// SIMATIC S7-200 SMART project (STEP 7-Micro/WIN SMART), CPU SR20

SYMBOL_TABLE 表格 1
搅拌1T定时器          C0
循环定时器            C1
任务阶段             VW10     // 当前任务阶段
提示注肥量            VW12
搅拌时长1T           VW14
目标液位1T           VW16     // 1T注水液位
当前液位1T           VW18
目标液位3T           VW20
当前液位3T           VW22
循环时长             VW24
运输完成标志1T到3T      VW26     // 启动运输前需要上位机置0
循环完成标志           VW28     // 循环前需要上位机清零
排污完成标志           VW30     // 排污前需要上位机清零
排污时长             VW32
水表               VW34
END_SYMBOL_TABLE

SYMBOL_TABLE 系统符号
Always_On        SM0.0    // 始终接通
First_Scan_On    SM0.1    // 仅在第一个扫描周期时接通
Clock_60s        SM0.4    // 针对 1 分钟的周期时间，时钟脉冲接通 30 s，断开 30 s.
END_SYMBOL_TABLE

ORGANIZATION_BLOCK MAIN:OB1
TITLE=注肥功能
BEGIN
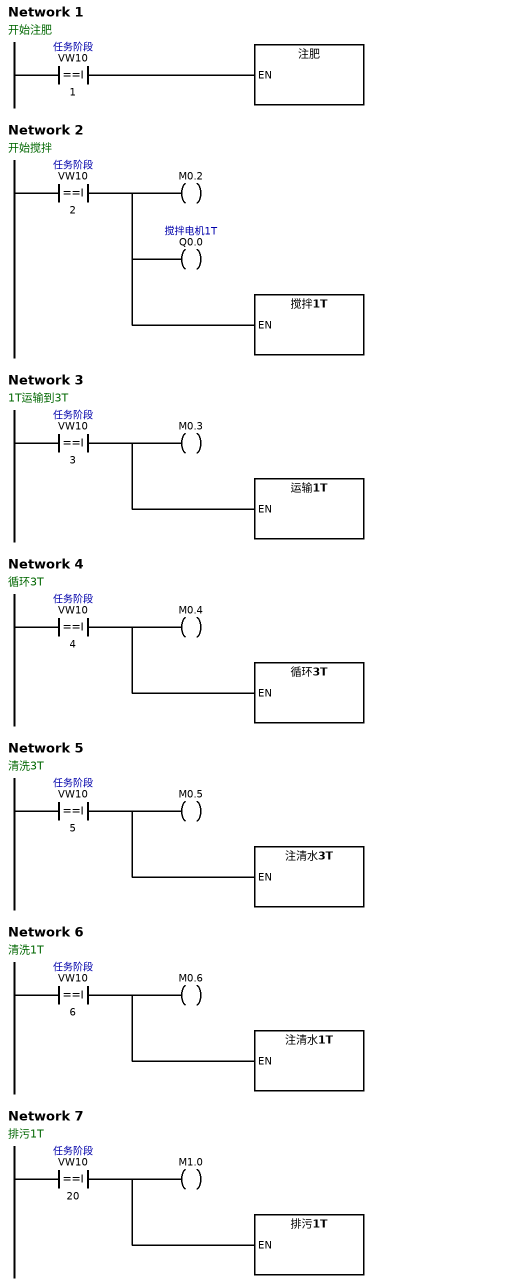
Network 1
// 开始注肥
LDW=   任务阶段:VW10, 1
CALL   注肥:SBR0
Network 2
// 开始搅拌
LDW=   任务阶段:VW10, 2
=      M0.2
=      搅拌电机1T:Q0.0
CALL   搅拌1T:SBR1
Network 3
// 1T运输到3T
LDW=   任务阶段:VW10, 3
=      M0.3
CALL   运输1T:SBR2
Network 4
// 循环3T
LDW=   任务阶段:VW10, 4
=      M0.4
CALL   循环3T:SBR4
Network 5
// 清洗3T
LDW=   任务阶段:VW10, 5
=      M0.5
CALL   注清水3T:SBR6
Network 6
// 清洗1T
LDW=   任务阶段:VW10, 6
=      M0.6
CALL   注清水1T:SBR7
Network 7
// 排污1T
LDW=   任务阶段:VW10, 20
=      M1.0
CALL   排污1T:SBR3
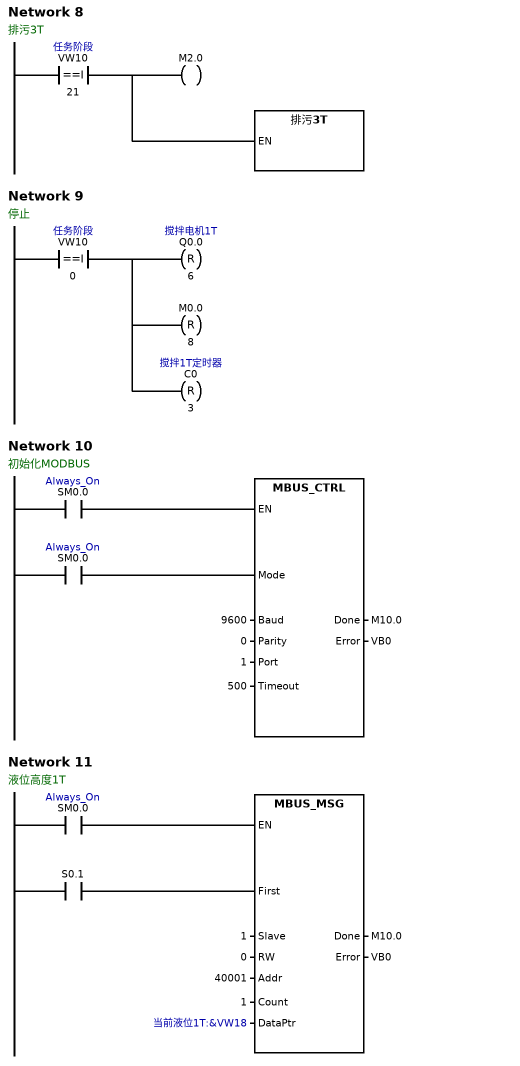
Network 8
// 排污3T
LDW=   任务阶段:VW10, 21
=      M2.0
CALL   排污3T:SBR5
Network 9
// 停止
LDW=   任务阶段:VW10, 0
R      搅拌电机1T:Q0.0, 6
R      M0.0, 8
R      搅拌1T定时器:C0, 3
Network 10
// 初始化MODBUS
LD     Always_On:SM0.0
=      L60.0
LD     Always_On:SM0.0
=      L63.7
LD     L60.0
CALL   MBUS_CTRL:SBR8, L63.7, 9600, 0, 1, 500, M10.0, VB0
Network 11
// 液位高度1T
LD     Always_On:SM0.0
=      L60.0
LD     S0.1
=      L63.7
LD     L60.0
CALL   MBUS_MSG:SBR9, L63.7, 1, 0, 40001, 1, &当前液位1T:VW18, M10.0, VB0
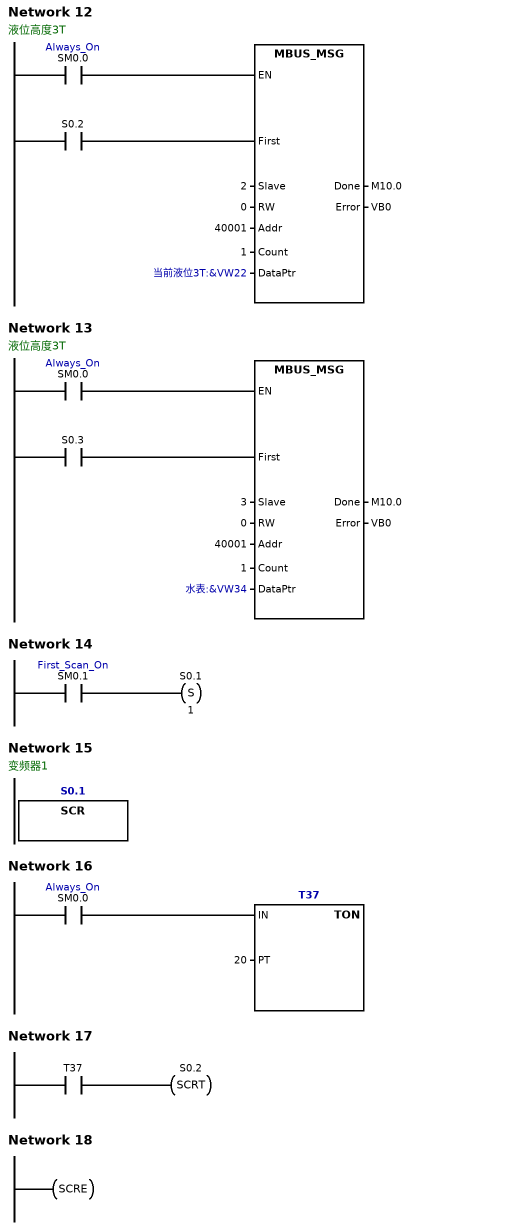
Network 12
// 液位高度3T
LD     Always_On:SM0.0
=      L60.0
LD     S0.2
=      L63.7
LD     L60.0
CALL   MBUS_MSG:SBR9, L63.7, 2, 0, 40001, 1, &当前液位3T:VW22, M10.0, VB0
Network 13
// 液位高度3T
LD     Always_On:SM0.0
=      L60.0
LD     S0.3
=      L63.7
LD     L60.0
CALL   MBUS_MSG:SBR9, L63.7, 3, 0, 40001, 1, &水表:VW34, M10.0, VB0
Network 14
LD     First_Scan_On:SM0.1
S      S0.1, 1
Network 15
// 变频器1
LSCR   S0.1
Network 16
LD     Always_On:SM0.0
TON    T37, 20
Network 17
LD     T37
SCRT   S0.2
Network 18
SCRE
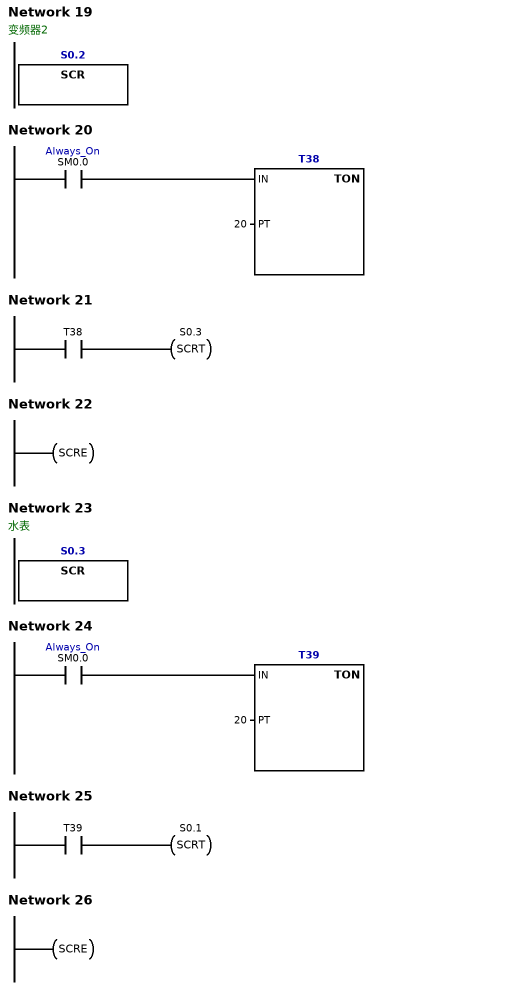
Network 19
// 变频器2
LSCR   S0.2
Network 20
LD     Always_On:SM0.0
TON    T38, 20
Network 21
LD     T38
SCRT   S0.3
Network 22
SCRE
Network 23
// 水表
LSCR   S0.3
Network 24
LD     Always_On:SM0.0
TON    T39, 20
Network 25
LD     T39
SCRT   S0.1
Network 26
SCRE
END_ORGANIZATION_BLOCK

SUBROUTINE_BLOCK 注肥:SBR0
TITLE=任务阶段1
BEGIN
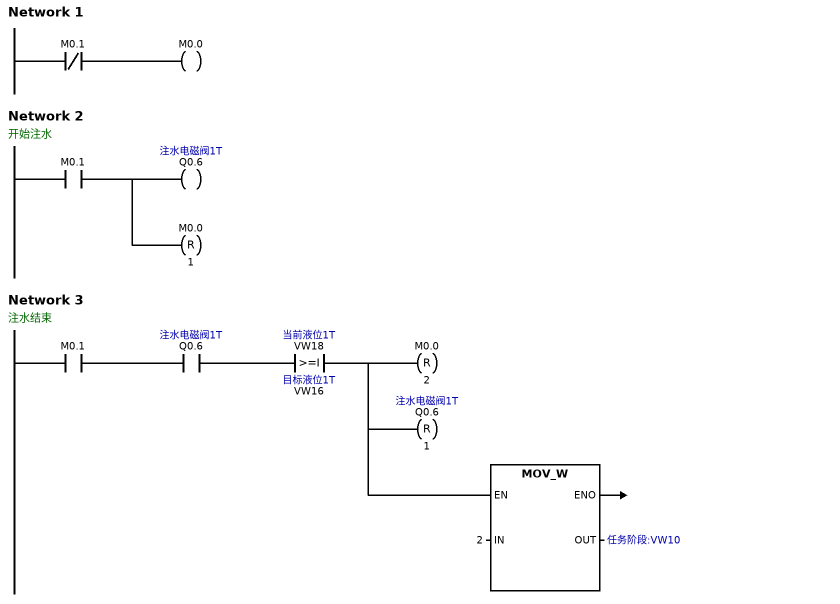
Network 1
LDN    M0.1
=      M0.0
Network 2
// 开始注水
LD     M0.1
=      注水电磁阀1T:Q0.6
R      M0.0, 1
Network 3
// 注水结束
LD     M0.1
A      注水电磁阀1T:Q0.6
AW>=   当前液位1T:VW18, 目标液位1T:VW16
R      M0.0, 2
R      注水电磁阀1T:Q0.6, 1
MOVW   2, 任务阶段:VW10
END_SUBROUTINE_BLOCK

SUBROUTINE_BLOCK 搅拌1T:SBR1
TITLE=任务阶段2
BEGIN
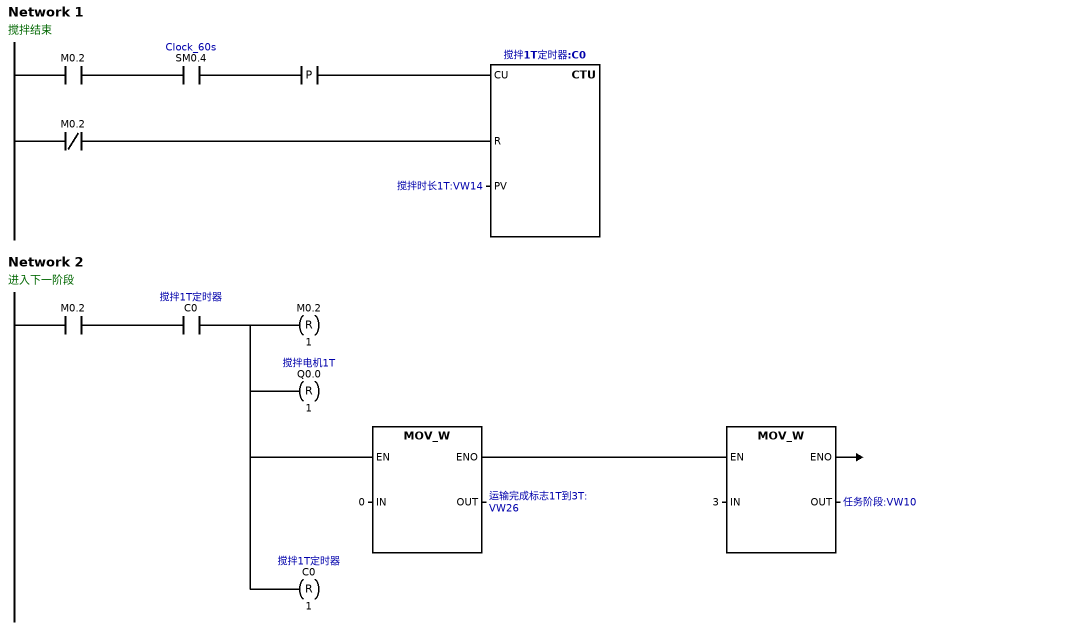
Network 1
// 搅拌结束
LD     M0.2
A      Clock_60s:SM0.4
EU
LDN    M0.2
CTU    搅拌1T定时器:C0, 搅拌时长1T:VW14
Network 2
// 进入下一阶段
LD     M0.2
A      搅拌1T定时器:C0
LPS
R      M0.2, 1
R      搅拌电机1T:Q0.0, 1
MOVW   0, 运输完成标志1T到3T:VW26
AENO
MOVW   3, 任务阶段:VW10
LPP
R      搅拌1T定时器:C0, 1
END_SUBROUTINE_BLOCK

SUBROUTINE_BLOCK 运输1T:SBR2
TITLE=任务阶段3
BEGIN
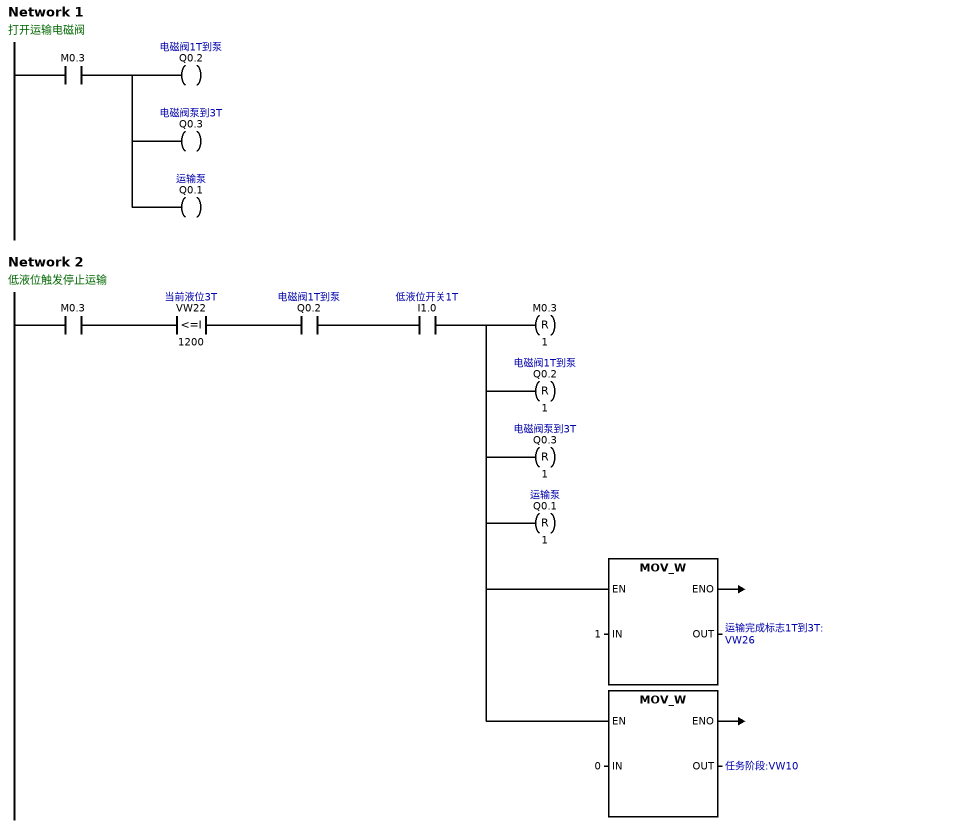
Network 1
// 打开运输电磁阀
LD     M0.3
=      电磁阀1T到泵:Q0.2
=      电磁阀泵到3T:Q0.3
=      运输泵:Q0.1
Network 2
// 低液位触发停止运输
LD     M0.3
AW<=   当前液位3T:VW22, 1200
A      电磁阀1T到泵:Q0.2
A      低液位开关1T:I1.0
R      M0.3, 1
R      电磁阀1T到泵:Q0.2, 1
R      电磁阀泵到3T:Q0.3, 1
R      运输泵:Q0.1, 1
MOVW   1, 运输完成标志1T到3T:VW26
MOVW   0, 任务阶段:VW10
END_SUBROUTINE_BLOCK

SUBROUTINE_BLOCK 排污1T:SBR3
TITLE=任务阶段20
BEGIN
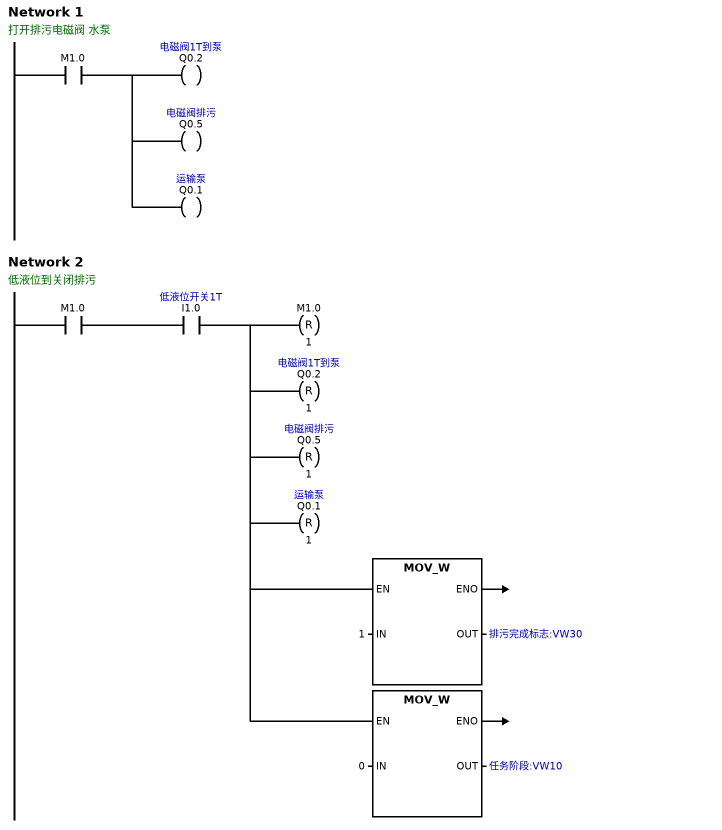
Network 1
// 打开排污电磁阀 水泵
LD     M1.0
=      电磁阀1T到泵:Q0.2
=      电磁阀排污:Q0.5
=      运输泵:Q0.1
Network 2
// 低液位到关闭排污
LD     M1.0
A      低液位开关1T:I1.0
R      M1.0, 1
R      电磁阀1T到泵:Q0.2, 1
R      电磁阀排污:Q0.5, 1
R      运输泵:Q0.1, 1
MOVW   1, 排污完成标志:VW30
MOVW   0, 任务阶段:VW10
END_SUBROUTINE_BLOCK

SUBROUTINE_BLOCK 循环3T:SBR4
TITLE=3T桶循环
BEGIN
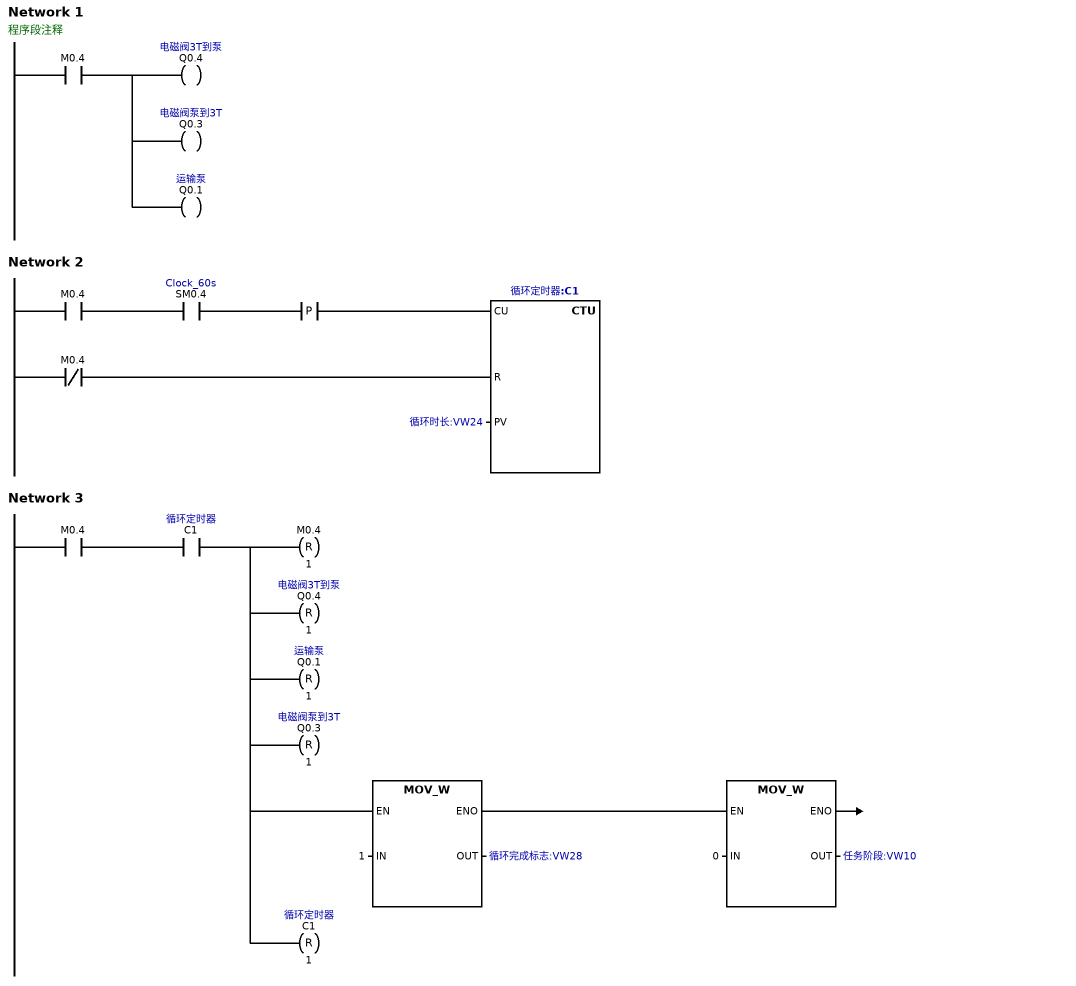
Network 1
// 程序段注释
LD     M0.4
=      电磁阀3T到泵:Q0.4
=      电磁阀泵到3T:Q0.3
=      运输泵:Q0.1
Network 2
LD     M0.4
A      Clock_60s:SM0.4
EU
LDN    M0.4
CTU    循环定时器:C1, 循环时长:VW24
Network 3
LD     M0.4
A      循环定时器:C1
LPS
R      M0.4, 1
R      电磁阀3T到泵:Q0.4, 1
R      运输泵:Q0.1, 1
R      电磁阀泵到3T:Q0.3, 1
MOVW   1, 循环完成标志:VW28
AENO
MOVW   0, 任务阶段:VW10
LPP
R      循环定时器:C1, 1
END_SUBROUTINE_BLOCK

SUBROUTINE_BLOCK 排污3T:SBR5
TITLE=任务阶段21
BEGIN
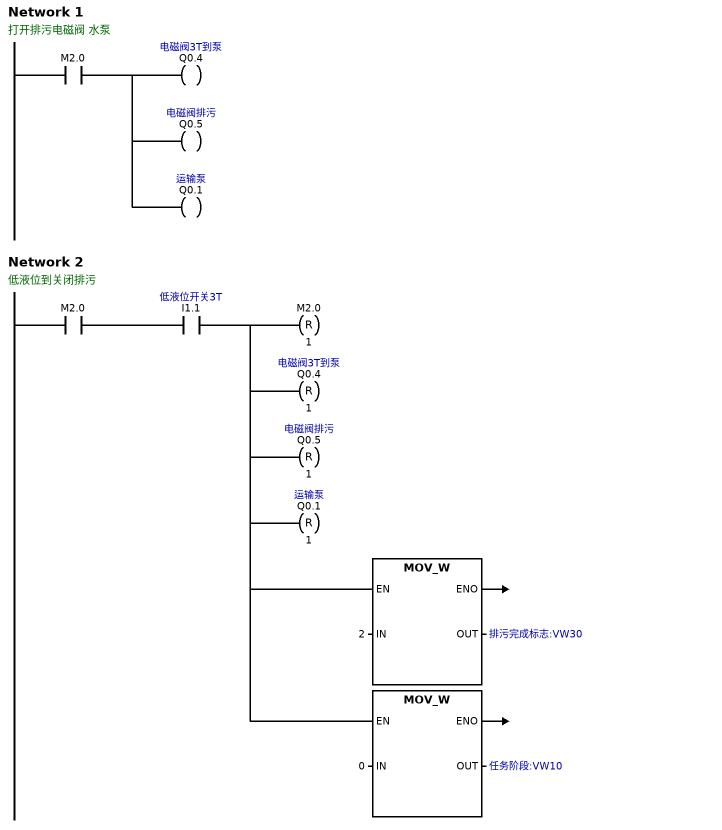
Network 1
// 打开排污电磁阀 水泵
LD     M2.0
=      电磁阀3T到泵:Q0.4
=      电磁阀排污:Q0.5
=      运输泵:Q0.1
Network 2
// 低液位到关闭排污
LD     M2.0
A      低液位开关3T:I1.1
R      M2.0, 1
R      电磁阀3T到泵:Q0.4, 1
R      电磁阀排污:Q0.5, 1
R      运输泵:Q0.1, 1
MOVW   2, 排污完成标志:VW30
MOVW   0, 任务阶段:VW10
END_SUBROUTINE_BLOCK

SUBROUTINE_BLOCK 注清水3T:SBR6
TITLE=子程序注释
BEGIN
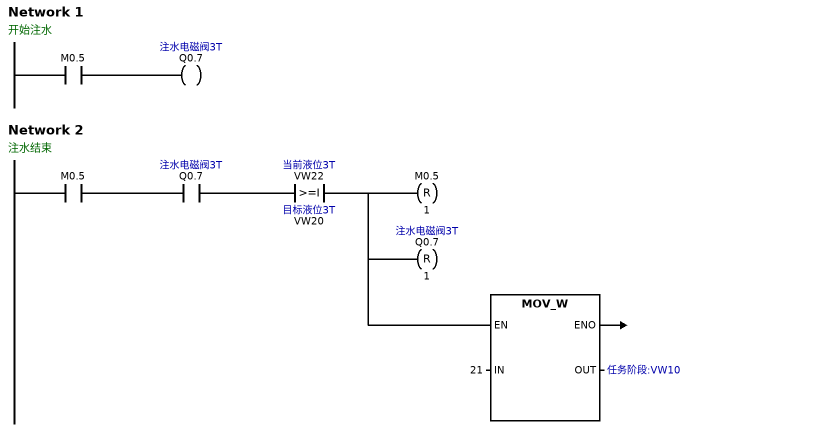
Network 1
// 开始注水
LD     M0.5
=      注水电磁阀3T:Q0.7
Network 2
// 注水结束
LD     M0.5
A      注水电磁阀3T:Q0.7
AW>=   当前液位3T:VW22, 目标液位3T:VW20
R      M0.5, 1
R      注水电磁阀3T:Q0.7, 1
MOVW   21, 任务阶段:VW10
END_SUBROUTINE_BLOCK

SUBROUTINE_BLOCK 注清水1T:SBR7
TITLE=子程序注释
BEGIN
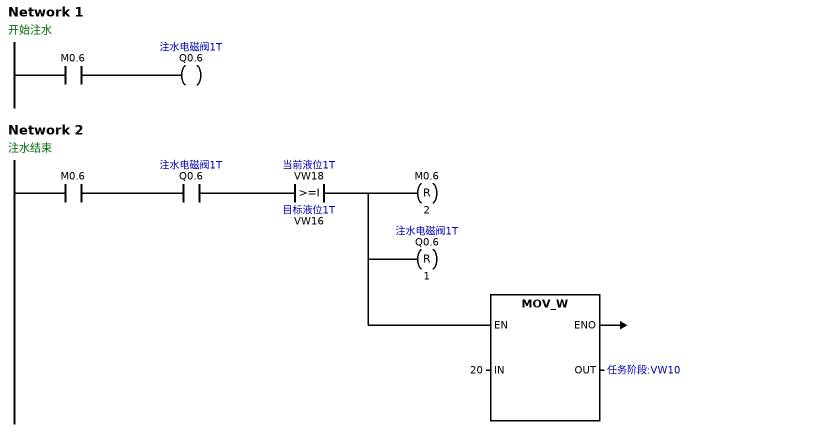
Network 1
// 开始注水
LD     M0.6
=      注水电磁阀1T:Q0.6
Network 2
// 注水结束
LD     M0.6
A      注水电磁阀1T:Q0.6
AW>=   当前液位1T:VW18, 目标液位1T:VW16
R      M0.6, 2
R      注水电磁阀1T:Q0.6, 1
MOVW   20, 任务阶段:VW10
END_SUBROUTINE_BLOCK

// SBR8: protected block, not included

// SBR9: protected block, not included

// SBR10: protected block, not included

DATA_BLOCK_TAB 页面_1
BEGIN
//数据页注释
//按 F1 获取帮助和示例数据页
         循环时长, 10
         搅拌时长1T, 30
END_DATA_BLOCK_TAB
